KUKA KRL data list: wkz1_ok.dat

&ACCESS RVP
&COMMENT CHK_TCP_C1
&PARAM DISKPATH = Program/FUNCIONANDO
DEFDAT  wkz1_ok
;FOLD EXTERNAL DECLARATIONS;%{PE}%MKUKATPBASIS,%CEXT,%VCOMMON,%P
;FOLD BASISTECH EXT;%{PE}%MKUKATPBASIS,%CEXT,%VEXT,%P
EXT  BAS (BAS_COMMAND  :IN,REAL  :IN )
DECL INT SUCCESS
;ENDFOLD (BASISTECH EXT)
;FOLD USER EXT;%{E}%MKUKATPUSER,%CEXT,%VEXT,%P
;Make your modifications here
;ENDFOLD (USER EXT)
;ENDFOLD (EXTERNAL DECLARATIONS)

;# ============ START PATH : wkz1_ok =============
DECL FDAT Fnew_wkz1_ok_p1={TOOL_NO 1,BASE_NO 0,IPO_FRAME #BASE,POINT2[] " "}
DECL PDAT PP_OLP1={VEL 100.0,ACC 50.0,APO_DIST 0.0}
DECL E6POS Xnew_wkz1_ok_p1={X 291.243988,Y -1285.88794,Z 233.281006,A 13.0198002,B 2.4052,C 1.18589997,S 2,T 10}
DECL FDAT Fnew_wkz1_ok_p2={TOOL_NO 1,BASE_NO 0,IPO_FRAME #BASE,POINT2[] " "}
DECL PDAT PP_OLP2={VEL 100.0,ACC 50.0,APO_DIST 0.0}
DECL E6POS Xnew_wkz1_ok_p2={X -473.602997,Y -1280.02002,Z -74.2460022,A 146.021698,B -0.95389998,C -2.53250003,S 2,T 2}
DECL FDAT Fnew_wkz1_ok_p3={TOOL_NO 1,BASE_NO 0,IPO_FRAME #BASE,POINT2[] " "}
DECL E6POS Xnew_wkz1_ok_p3={X -886.51001,Y -1289.66003,Z 13.3669996,A 171.756897,B -2.65339994,C -0.53549999,S 2,T 2}
DECL LDAT LL_OLP1={VEL 2.0,ACC 100.0,APO_DIST 0.0,APO_FAC 0.0,ORI_TYP #VAR,CIRC_TYP #BASE,JERK_FAC 50.0}
DECL FDAT Fnew_wkz1_ok_ptcpc={TOOL_NO 1,BASE_NO 0,IPO_FRAME #BASE,POINT2[] " "}
DECL E6POS Xnew_wkz1_ok_ptcpc={X -881.550415,Y -1291.69397,Z 47.3409119,A 171.412704,B -2.65365791,C -0.829671085,S 18,T 2,E1 0.0,E2 0.0,E3 0.0,E4 0.0,E5 0.0,E6 0.0}
DECL LDAT LL_OLP2={VEL 2.0,ACC 100.0,APO_DIST 0.0,APO_FAC 0.0,ORI_TYP #VAR,CIRC_TYP #BASE,JERK_FAC 50.0}
DECL FDAT Fnew_wkz1_ok_p4={TOOL_NO 1,BASE_NO 0,IPO_FRAME #BASE,POINT2[] " "}
DECL E6POS Xnew_wkz1_ok_p4={X -886.51001,Y -1289.66003,Z 13.3669996,A 171.756897,B -2.65339994,C -0.53549999,S 2,T 2}
DECL LDAT LL_OLP3={VEL 2.0,ACC 100.0,APO_DIST 0.0,APO_FAC 0.0,ORI_TYP #VAR,CIRC_TYP #BASE,JERK_FAC 50.0}
DECL FDAT Fnew_wkz1_ok_p5={TOOL_NO 1,BASE_NO 0,IPO_FRAME #BASE,POINT2[] " "}
DECL PDAT PP_OLP3={VEL 100.0,ACC 50.0,APO_DIST 0.0}
DECL E6POS Xnew_wkz1_ok_p5={X -473.602997,Y -1280.02002,Z -74.2460022,A 146.021698,B -0.95389998,C -2.53250003,S 2,T 2}
DECL FDAT Fnew_wkz1_ok_p6={TOOL_NO 1,BASE_NO 0,IPO_FRAME #BASE,POINT2[] " "}
DECL PDAT PP_OLP4={VEL 100.0,ACC 50.0,APO_DIST 0.0}
DECL E6POS Xnew_wkz1_ok_p6={X 291.243988,Y -1285.88794,Z 233.281006,A 13.0198002,B 2.4052,C 1.18589997,S 2,T 10}
ENDDAT
